// TwinCAT 3 PLC project PLC
// ProgramVersion: 3.1.4024.0
// libraries:
//   Tc2_EtherCAT, * (Beckhoff Automation GmbH)
//   Tc2_MDP, * (Beckhoff Automation GmbH)
//   Tc2_Standard, * (Beckhoff Automation GmbH)
//   Tc2_System, * (Beckhoff Automation GmbH)
//   Tc2_Utilities, * (Beckhoff Automation GmbH)
//   Tc3_JsonXml, * (Beckhoff Automation GmbH)
//   Tc3_Module, * (Beckhoff Automation GmbH)
//   Util, * (System)
// project tree:
//   DUTs/ EtherCAT_Offline_Config.TcDUT, E_Variant.TcDUT
//   GVLs/ GVL.TcGVL
//   / PlcTask.TcTTO
//   POUs/ MAIN.TcPOU, PRG_CheckEtherCATTopology.TcPOU, PRG_SwapBootFolder.TcPOU
// real-time tasks:
//   TASK PlcTask: cycle T#4ms, priority 20, ADS port 350
// I/O:
//   DEVICE Device 1 (EtherCAT), AmsNetId 0.0.0.0.2.1
//     Term 1 (EK1100) [EK1100 EtherCAT Coupler (2A E-Bus)]
//       Term 2 (EL2809) [EL2809 16Ch. Dig. Output 24V, 0.5A] (disabled)
//       Term 2 (EL2809-0015) [EL2809-0015 16Ch. Dig. Output 24V DC, 0.35A, not short-circuit proof] (disabled)
// variable links:
//   __THIS__ <-> Device 1 (EtherCAT)
//     PlcTask Inputs/PRG_CheckEtherCATTopology.EcMasterNetID <-> InfoData/AmsNetId
//   __THIS__ <-> Device 1 (EtherCAT)/Term 1 (EK1100)/Term 2 (EL2809)
//     PlcTask Outputs/MAIN.Outputs[{0..15}] <-> Channel {1..16}/Output  (16 links)
//   __THIS__ <-> Device 1 (EtherCAT)/Term 1 (EK1100)/Term 2 (EL2809-0015)
//     PlcTask Outputs/MAIN.Outputs[{0..15}] <-> Channel {1..16}/Output  (16 links)
//   PLC Instance <-> Device 1 (EtherCAT)
//     PlcTask Inputs/PRG_CheckEtherCATTopology.EcMasterNetID <-> InfoData/AmsNetId
//   PLC Instance <-> Device 1 (EtherCAT)/Term 1 (EK1100)/Term 2 (EL2809)
//     PlcTask Outputs/MAIN.Outputs[{0..15}] <-> Channel {1..16}/Output  (16 links)

CONFIGURATION PLC
    RESOURCE PLC ON TwinCAT3
        TASK PlcTask(INTERVAL := T#4ms, PRIORITY := 20);
        PROGRAM MAIN WITH PlcTask : MAIN;
    END_RESOURCE
END_CONFIGURATION

// ---- DUTs/EtherCAT_Offline_Config.TcDUT
TYPE
    EtherCAT_Offline_Config : ARRAY[1..GVL.MaxNumOfSlaves] OF ST_EcSlaveConfigData;
END_TYPE

// ---- DUTs/E_Variant.TcDUT
{attribute 'qualified_only'}
{attribute 'to_string'}
TYPE
    E_Variant :
    (
        Unknown := 0,
        RevA    := 1,
        RevB    := 2,
        End     := 3
    );
END_TYPE

// ---- GVLs/GVL.TcGVL
VAR_GLOBAL CONSTANT
    {IF defined (RevA)}
    CurrentVariant : E_Variant := E_Variant.RevA;
    {ELSIF defined (RevB)}
    CurrentVariant : E_Variant := E_Variant.RevB;
    {ELSE}
    CurrentVariant : E_Variant := E_Variant.Unknown;
    {END_IF}
    MaxNumOfSlaves : UINT := 5;
END_VAR
VAR_GLOBAL
    sCurrentVariant : T_MaxString := TO_STRING(CurrentVariant);
END_VAR

// ---- POUs/MAIN.TcPOU
PROGRAM MAIN
VAR
    Outputs AT %Q* : ARRAY[0..15] OF BOOL;
    fbBlink        : BLINK;
    i              : UDINT;
	
	xCheckTopologyForVariantMatch :BOOL:=TRUE;
	xSwapBootFolder	:BOOL;

END_VAR

fbBlink(ENABLE := TRUE, TIMELOW := T#1S, TIMEHIGH := T#1S);

FOR i := 0 TO 15 DO
    Outputs[i] := fbBlink.OUT;
END_FOR



PRG_CheckEtherCATTopology(
	xCheckTopology:=xCheckTopologyForVariantMatch , 
	eMatchedVariant=> , 
	sMatchedVariant=> , 
	xScanAndConfigMatch=> , 
	xMoreThanOnMatch=> , 
	bBusy=> , 
	bError=> , 
	nErrorID=> , 
	ErrorOnStep=> );

PRG_SwapBootFolder(
	VariantToLoad:=PRG_CheckEtherCATTopology.eMatchedVariant , 
	xSwapBootFolder:=xSwapBootFolder , 
	busy=> , 
	error=> , 
	ErrorID=> );

END_PROGRAM

// ---- POUs/PRG_CheckEtherCATTopology.TcPOU
//Each vairent needs to be run once, for this to work properly - the configured ethercat devices are stored in a JSON file at %TC_RESOURCEPATH% VariantName.json'
PROGRAM PRG_CheckEtherCATTopology
VAR_INPUT
    xCheckTopology : BOOL := TRUE;
END_VAR
VAR
    rtCheck              : R_TRIG;
    EcMasterNetID AT %I* : AMSNETID;
    fbEcGetConfSlaves    : FB_EcGetConfSlaves;
    fbEcGetScannedSlaves : FB_EcGetScannedSlaves;

    CurrentEcConfSlaveInfo : EtherCAT_Offline_Config;                               //: ARRAY[0..EC_MAX_SLAVES] OF ST_EcSlaveConfigData;
    ArrEcScannedSlaveInfo  : ARRAY[1..GVL.MaxNumOfSlaves] OF ST_EcSlaveScannedData; //: ARRAY[0..EC_MAX_SLAVES] OF ST_EcSlaveScannedData;
    i                      : UINT;

    eStep : (Init,
        GetOffLineConfig,
        GenerateCurrentVarientEcConfigFile,
        SavingActiveVarient,
        LoadVariantXEcConfigFiles,
        GetOnLineScanned,
        compare);

    //Description of all available varients.
    arVarientEcConfig : ARRAY[E_Variant.Unknown..E_Variant.End] OF EtherCAT_Offline_Config;

    //File handling - store ethercat configuration into a file outside of the boot folder
    Result            : HRESULT;
    fbJson            : FB_JsonSaxWriter;
    fbJsonDataType    : FB_JsonReadWriteDataType;
    fbJsonFileHandler : FB_JsonDomParser;
    bSave             : BOOL;
    bSaved            : BOOL;
    bLoad             : BOOL;
    bLoaded           : BOOL;
    eVariantIndex     : E_Variant;
    aVariantIsTheSame : ARRAY[E_Variant.Unknown..E_Variant.End] OF BOOL;

    sFilePath : STRING(255);
    sJsonDoc  : STRING(10000);

    fbformat : FB_FormatString2;
    sFormat  : T_MaxString;
    sOut     : STRING(600);
END_VAR
VAR_OUTPUT
    eMatchedVariant     : E_Variant;
    sMatchedVariant     : T_MaxString;
    xScanAndConfigMatch : BOOL;
    xMoreThanOnMatch    : BOOL;

    bBusy       : BOOL;
    bError      : BOOL;
    nErrorID    : UDINT;
    ErrorOnStep : DINT;
END_VAR

rtCheck(CLK := xCheckTopology);

CASE eStep OF

    Init:
        bBusy := FALSE;

        IF rtCheck.q THEN
            eMatchedVariant  := E_Variant.Unknown;
            sMatchedVariant  := '';
            xMoreThanOnMatch := FALSE;
            bBusy            := TRUE;
            bError           := FALSE;
            nErrorID         := 0;
            eStep            := GetOffLineConfig;
        END_IF

    GetOffLineConfig:
        fbEcGetConfSlaves(sNetId := F_CreateAmsNetId(EcMasterNetID),
            pArrEcConfSlaveInfo := ADR(CurrentEcConfSlaveInfo),
            cbBufLen := SIZEOF(CurrentEcConfSlaveInfo),
            bExecute := TRUE);

        IF NOT fbEcGetConfSlaves.bBusy THEN
            fbEcGetConfSlaves(bExecute := FALSE);

            IF NOT fbEcGetConfSlaves.bError THEN
                eStep := GenerateCurrentVarientEcConfigFile;
            ELSE
                bError      := TRUE;
                nErrorID    := fbEcGetConfSlaves.nErrorID;
                ErrorOnStep := eStep;
                eStep       := Init;
                ADSLOGSTR(ADSLOG_MSGTYPE_ERROR OR ADSLOG_MSGTYPE_LOG, 'error %s getting configured EtherCAT slaves', TO_STRING(nErrorID));
            END_IF
        END_IF

    GenerateCurrentVarientEcConfigFile:

        fbJson.ResetDocument();

        fbJsonDataType.AddJsonValueFromSymbol(fbWriter := fbJson,
            sDatatype := 'EtherCAT_Offline_Config',
            nData := SIZEOF(CurrentEcConfSlaveInfo),
            pData := ADR(CurrentEcConfSlaveInfo),
            hrErrorCode => Result);

        IF Result <> S_OK THEN
            bError      := TRUE;
            nErrorID    := TO_UDINT(Result);
            ErrorOnStep := eStep;
            eStep       := Init;
            ADSLOGSTR(ADSLOG_MSGTYPE_ERROR OR ADSLOG_MSGTYPE_LOG, 'error %s getting json value from Symbol', TO_STRING(Result));
            RETURN;
        END_IF

        fbJson.CopyDocument(pDoc := sJsonDoc, nDoc := SIZEOF(sJsonDoc), hrErrorCode => Result);

        IF Result <> S_OK THEN
            bError      := TRUE;
            nErrorID    := TO_UDINT(Result);
            ErrorOnStep := eStep;
            eStep       := Init;
            ADSLOGSTR(ADSLOG_MSGTYPE_ERROR OR ADSLOG_MSGTYPE_LOG, 'error %s copying json document', TO_STRING(Result));
            RETURN;
        END_IF

        fbJsonFileHandler.ParseDocument(sJson := sJsonDoc);

        sFilePath := CONCAT('%TC_RESOURCEPATH%', CONCAT(TO_STRING(GVL.CurrentVariant), '.json'));

        bSave := TRUE;
        eStep := SavingActiveVarient;

    SavingActiveVarient:
        IF bSave THEN
            bSaved := fbJsonFileHandler.SaveDocumentToFile(sFilePath, bSave);
        END_IF

        IF NOT bSave THEN
            IF bSaved THEN
                eStep         := LoadVariantXEcConfigFiles;
                bLoad         := TRUE;
                eVariantIndex := E_Variant.Unknown + 1;
            ELSE
                ErrorOnStep := eStep;
                eStep       := Init;
                ADSLOGSTR(ADSLOG_MSGTYPE_ERROR OR ADSLOG_MSGTYPE_LOG, 'error saving file %s', sFilePath);
                RETURN;
            END_IF
        END_IF

    LoadVariantXEcConfigFiles:
        sFilePath := CONCAT('%TC_RESOURCEPATH%', CONCAT(TO_STRING(eVariantIndex), '.json'));

        IF bLoad THEN
            bLoaded := fbJsonFileHandler.LoadDocumentFromFile(sFilePath, bLoad);
        END_IF

        IF NOT bLoad THEN
            IF bLoaded THEN
                fbJsonFileHandler.CopyDocument(pDoc := sJsonDoc, nDoc := SIZEOF(sJsonDoc));
                fbJsonDataType.SetSymbolFromJson(sJson := sJsonDoc,
                    sDatatype := 'EtherCAT_Offline_Config',
                    nData := SIZEOF(arVarientEcConfig[eVariantIndex]),
                    pData := ADR(arVarientEcConfig[eVariantIndex]),
                    hrErrorCode => Result);

                IF Result = S_OK THEN
                    IF eVariantIndex = E_Variant.End - 1 THEN
                        eStep := GetOnLineScanned;
                    ELSE
                        bLoad         := TRUE;
                        eVariantIndex := eVariantIndex + 1;
                    END_IF
                ELSE
                    bError      := TRUE;
                    nErrorID    := TO_UDINT(Result);
                    ErrorOnStep := eStep;
                    eStep       := Init;
                    ADSLOGSTR(ADSLOG_MSGTYPE_ERROR OR ADSLOG_MSGTYPE_LOG, 'error %s set symbol from json', TO_STRING(Result));
                    RETURN;
                END_IF
            ELSE
                ADSLOGSTR(ADSLOG_MSGTYPE_ERROR OR ADSLOG_MSGTYPE_LOG, 'Error loading file %s', sFilePath);
                bError      := TRUE;
                ErrorOnStep := eStep;
                eStep       := Init;
            END_IF
        END_IF

    GetOnLineScanned:
        fbEcGetScannedSlaves(bExecute := TRUE,
            sNetId := F_CreateAmsNetId(EcMasterNetID),
            pArrEcScannedSlaveInfo := ADR(ArrEcScannedSlaveInfo),
            cbBufLen := SIZEOF(ArrEcScannedSlaveInfo));

        IF NOT fbEcGetScannedSlaves.bBusy THEN
            fbEcGetScannedSlaves(bExecute := FALSE);

            IF NOT fbEcGetScannedSlaves.bError THEN
                eStep := compare;
            ELSE
                bError      := TRUE;
                nErrorID    := fbEcGetScannedSlaves.nErrorId;
                ErrorOnStep := eStep;
                eStep       := Init;
                ADSLOGSTR(ADSLOG_MSGTYPE_ERROR OR ADSLOG_MSGTYPE_LOG, 'error % getting scanned EtherCAT slaves', TO_STRING(nErrorID));
            END_IF
        END_IF

    compare:
        //This compare operation might be over complex for most cases. Here every device in the network is checked to see if the EtherCAT slave VPR (vendor, product, and revision) matchs the offline configuration, and online found devices. 
        //It might be sutiable to only check one specfic slave location.	

        //Checks if the current scaned devices matchs the configured devices
        xScanAndConfigMatch := TRUE;

        FOR i := 1 TO GVL.MaxNumOfSlaves DO
            IF ArrEcScannedSlaveInfo[i].stSlaveIdentity.vendorId <> CurrentEcConfSlaveInfo[i].stSlaveIdentity.vendorId OR
                ArrEcScannedSlaveInfo[i].stSlaveIdentity.productCode <> CurrentEcConfSlaveInfo[i].stSlaveIdentity.productCode OR
                ArrEcScannedSlaveInfo[i].stSlaveIdentity.revisionNo <> CurrentEcConfSlaveInfo[i].stSlaveIdentity.revisionNo
                THEN
                xScanAndConfigMatch := FALSE;
            END_IF
        END_FOR

        IF xScanAndConfigMatch THEN
            ADSLOGSTR(ADSLOG_MSGTYPE_HINT OR ADSLOG_MSGTYPE_LOG, 'The current EtherCAT configuration matchs the scanned devices', '');
        END_IF

        //Check all variants against what was found
        MEMSET(ADR(aVariantIsTheSame), 1, SIZEOF(aVariantIsTheSame));

        FOR eVariantIndex := E_Variant.Unknown TO E_Variant.End DO //Check against all variants
            FOR i := 1 TO GVL.MaxNumOfSlaves DO                    //Check the found slaves against a variant offline config
                IF ArrEcScannedSlaveInfo[i].stSlaveIdentity.vendorId <> arVarientEcConfig[eVariantIndex][i].stSlaveIdentity.vendorId OR
                    ArrEcScannedSlaveInfo[i].stSlaveIdentity.productCode <> arVarientEcConfig[eVariantIndex][i].stSlaveIdentity.productCode OR
                    ArrEcScannedSlaveInfo[i].stSlaveIdentity.revisionNo <> arVarientEcConfig[eVariantIndex][i].stSlaveIdentity.revisionNo
                    THEN
                    aVariantIsTheSame[eVariantIndex] := FALSE;
                END_IF
            END_FOR
        END_FOR

        FOR eVariantIndex := E_Variant.Unknown + 1 TO E_Variant.End - 1 DO
            IF aVariantIsTheSame[eVariantIndex] THEN
                IF eMatchedVariant = E_Variant.Unknown THEN
                    eMatchedVariant := eVariantIndex;
                    sMatchedVariant := TO_STRING(eMatchedVariant);
                ELSE
                    xMoreThanOnMatch := TRUE;
                    ADSLOGSTR(ADSLOG_MSGTYPE_WARN OR ADSLOG_MSGTYPE_LOG, 'more than one variant EtherCAT configuration matchs what was scanned', '');
                END_IF
            END_IF
        END_FOR

        IF eMatchedVariant <> E_Variant.Unknown AND NOT xMoreThanOnMatch AND NOT xScanAndConfigMatch THEN
            sFormat := 'The current EtherCAT configuration (variant %s) doesnt match what was scanned consider loading variant %s ';
            fbFormat(pFormatString := ADR(sFormat),
                arg1 := F_STRING(GVL.sCurrentVariant),
                arg2 := F_STRING(sMatchedVariant),
                pDstString := ADR(sOut),
                nDstSize := SIZEOF(sOut));

            ADSLOGSTR(ADSLOG_MSGTYPE_WARN OR ADSLOG_MSGTYPE_LOG, sOut, '');
        END_IF

        eStep := Init;

END_CASE

END_PROGRAM

// ---- POUs/PRG_SwapBootFolder.TcPOU
PROGRAM PRG_SwapBootFolder
VAR_INPUT
    VariantToLoad   : E_Variant;
    xSwapBootFolder : BOOL;
END_VAR
VAR
    ntCallPowerShellScript : NT_StartProcess;
END_VAR
VAR_OUTPUT
    busy    : BOOL;
    error   : BOOL;
    ErrorID : UDINT;
END_VAR

ntCallPowerShellScript(NETID := '',
    PATHSTR := 'C:\TwinCAT\3.1\Target\Resource\VariantSwitch.bat',
    DIRNAME := 'C:\TwinCAT\3.1\Target\Resource\',
    COMNDLINE := TO_STRING(VariantToLoad),
    START := xSwapBootFolder,
    TMOUT :=,
    BUSY => busy,
    ERR => error,
    ERRID => ErrorID);

END_PROGRAM
